Staubli VAL3: onExit.pgx

program onExit()
begin
  //
end
